// TIA Portal V21 export
FUNCTION_BLOCK "DATALOG TRIGGER BLOCK"   // FB11, LAD
{ S7_Optimized_Access := 'TRUE' }
// stored: MemoryReserve 100, SetENOAutomatically false
   VAR_INPUT
      "SET TIME" : Int;
      RESET : Bool;
      INPUT : Bool;
   END_VAR
   VAR_OUTPUT
      "PRESENT VALUE OF TIME" : Int;
      SEC : Int;
      DONE : Bool;
      "TRIGGER BIT" : Bool;
      "ALARM BIT" : Bool;
   END_VAR
   VAR
      "TIMER 1" { S7_SetPoint := 'True'} : IEC_TIMER;
   END_VAR
   VAR RETAIN
      "COUNTER1 0" { S7_SetPoint := 'True'} : IEC_COUNTER;
      "COUNTER1 1" { S7_SetPoint := 'True'} : IEC_COUNTER;
      TPULSE { S7_SetPoint := 'True'} : IEC_TIMER;
   END_VAR
   VAR_TEMP   // added for the SCL form of the ladder/FBD networks
      _w1 : Bool;
      _w2 : Bool;
   END_VAR
BEGIN

REGION Network 2
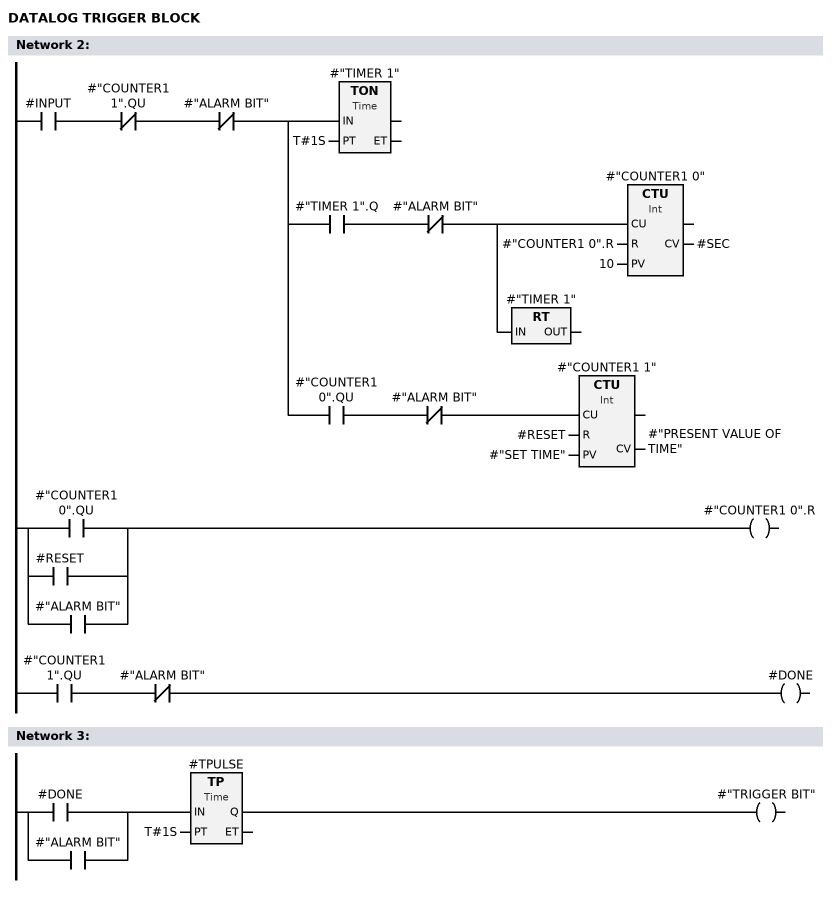
   RUNG wire#powerrail
      Contact( #INPUT )
      I_Contact( #"COUNTER1 1".QU )
      I_Contact( #"ALARM BIT" )
      wire#w1
      { S7_Templates := "time_type := Time" } #"TIMER 1".TON(pt := T#1S, et =>)
   END_RUNG
   RUNG wire#w1
      Contact( #"TIMER 1".Q )
      I_Contact( #"ALARM BIT" )
      wire#w2
      { S7_Templates := "value_type := Int" } #"COUNTER1 0".CTU(r := #"COUNTER1 0".R, pv := 10, cv => #SEC)
   END_RUNG
   RUNG wire#w2
      RT_Coil( #"TIMER 1" )
   END_RUNG
   RUNG wire#w1
      Contact( #"COUNTER1 0".QU )
      I_Contact( #"ALARM BIT" )
      { S7_Templates := "value_type := Int" } #"COUNTER1 1".CTU(r := #RESET, pv := #"SET TIME", cv => #"PRESENT VALUE OF TIME")
   END_RUNG
   RUNG wire#powerrail
      Contact( #"COUNTER1 0".QU )
      wire#w3
      Coil( #"COUNTER1 0".R )
   END_RUNG
   RUNG wire#powerrail
      Contact( #RESET )
   END_RUNG wire#w3
   RUNG wire#powerrail
      Contact( #"ALARM BIT" )
   END_RUNG wire#w3
   RUNG wire#powerrail
      Contact( #"COUNTER1 1".QU )
      I_Contact( #"ALARM BIT" )
      Coil( #DONE )
   END_RUNG
   // the same network as SCL:
   #_w1 := #INPUT AND NOT #"COUNTER1 1".QU AND NOT #"ALARM BIT";
   #"TIMER 1".TON(IN := #_w1, PT := T#1S);
   #_w2 := #_w1 AND #"TIMER 1".Q AND NOT #"ALARM BIT";
   #"COUNTER1 0".CTU(CU := #_w2, R := #"COUNTER1 0".R, PV := 10, CV => #SEC);
   IF #_w2 THEN RESET_TIMER(#"TIMER 1"); END_IF;
   #"COUNTER1 1".CTU(CU := #_w1 AND #"COUNTER1 0".QU AND NOT #"ALARM BIT",
                     R := #RESET,
                     PV := #"SET TIME",
                     CV => #"PRESENT VALUE OF TIME");
   #"COUNTER1 0".R := #"COUNTER1 0".QU OR #RESET OR #"ALARM BIT";
   #DONE := #"COUNTER1 1".QU AND NOT #"ALARM BIT";
END_REGION

REGION Network 3
   RUNG wire#powerrail
      Contact( #DONE )
      wire#w1
      { S7_Templates := "time_type := Time" } #TPULSE.TP(pt := T#1S, et =>)
      Coil( #"TRIGGER BIT" )
   END_RUNG
   RUNG wire#powerrail
      Contact( #"ALARM BIT" )
   END_RUNG wire#w1
   // the same network as SCL:
   #TPULSE.TP(IN := #DONE OR #"ALARM BIT", PT := T#1S);
   #"TRIGGER BIT" := #TPULSE.Q;
END_REGION
END_FUNCTION_BLOCK
